///Automatically generated by BoxConfigurator 
VAR_GLOBAL
	fbSG_001                : FB_ProBOXSG;
	fbSG_002                : FB_ProBOXSG;
END_VAR

(* stored: Version 1.1.0.1, ProductVersion 3.1.4024.9
   GVL Groups: Id {ded58393-b36c-4408-ae22-9cb4a48d6cc4} *)
